{attribute 'GeneratedUsingTerminal: EL5001-0000-1016'}
{attribute addProperty BoxType "EL5001-0000-1016"}
{attribute addProperty Description "EL5001 1Ch. SSI Encoder"}
{attribute addProperty Physics "KK"}
{attribute addProperty Id "Channel_1AT %I*Channel_DD2C734A5WcStateAT %I*WcState_9091E0EB2InfoDataAT %I*InfoData_32EB74EA10"}
{attribute addProperty CRC "2978392052"}
{attribute addProperty Size "17"}
TYPE EL5001_B186A7F4 EXTENDS EtcSlaveTerminalBase_947E5A46 :
STRUCT
	{attribute addProperty Name "Channel_1"}
	Channel_1 : Channel_DD2C734A;
	{attribute addProperty Name "WcState"}
	WcState : WcState_9091E0EB;
	{attribute addProperty Name "InfoData"}
	InfoData : InfoData_32EB74EA;
END_STRUCT
END_TYPE

(* stored: Version 1.2.0.0, ProductVersion 3.1.4024.11
   DUT EL5001_B186A7F4: Id {df0051c7-f80a-430f-aa16-e10afb9858b7} *)
